SUBAPPLICATION logiBUS_AI_Calibrate_3P_Subscribe_VT_OPC (* Remote-Subscribe eines bereits kalibrierten physikalischen Werts (M2M, von der Sensor-Station, 3-Punkt-Kalibrierung) -> VT-Anzeige (Q_NumericValue_PHYSA) + lokaler Re-Publish + optionaler CAL_OUT-Plug fuer lokale Consumer. Die physischen VT-Elemente bleiben hier (dort wo die VT ist): C_MIN/C_MID/C_MAX-Tasten rufen per CLIENT_0 direkt die ID_MIN_METHOD/ID_MID_TRIGGER_METHOD/ID_MAX_METHOD auf der Sensor-Station auf (logiBUS_AI_Calibrate_3P_IDA_OPC) - echter Event-zu-Event-Methodenaufruf, kein Toggle/Publish/Subscribe-Umweg. Die drei Referenzwert-Eingabefelder MIN/MID/MAX_REF (NumericValue_TO_AR2_OPC) werden weiterhin LOKAL publiziert und von der Sensor-Station remote abonniert - MID_REF/MAX_REF zusaetzlich als plain-AR-Plugs MIDREF_OUT/MAXREF_OUT re-exponiert (z.B. fuer Fuellband_Oben_Erkennung/Befuellautomatik). Ersetzt logiBUS_AI_Calibrate_3P_Remote_IDA_OPC: Kalibrierung selbst laeuft jetzt auf der Sensor-Station (logiBUS_AI_Calibrate_3P_IDA_OPC), hier bleibt nur noch Anzeige + VT-Bedienelemente-Weiterleitung. *)
  (* Standard: 61499-2; Description: Copyright (c) 2026 Meisterschulen am Ostbahnhof This program and the accompanying materials are made available under the terms of the Eclipse Public License 2.0 which is available at https://www.eclipse.org/legal/epl-2.0/ SPDX-License-Identifier: EPL-2.0 *)
  (* Version 1.0, 2026-09-18, Franz Höpfinger, Meisterschulen am Ostbahnhof, initial implementation - Analog-Lokal-Verarbeitung Phase 6 (Plan cuddly-bubbling-twilight): 3P-Pendant zu logiBUS_AI_Calibrated_Subscribe_VT_OPC (2P), fuer Fuellband Winkel (STG2). Plugs CAL_OUT/MIDREF_OUT/MAXREF_OUT 1:1 aus logiBUS_AI_Calibrate_3P_Remote_IDA_OPC uebernommen, damit bestehende Consumer (Fuellband_Oben_Erkennung, Befuellautomatik) unveraendert bleiben. *)
  PACKAGE MyLib::sys;
  IMPORT isobus::UT::Q::const::IDs::ID_NULL;
  IMPORT isobus::UT::io::Button::ButtonActivationCode::BT_PRESSED_LATCHED;
  IMPORT logiBUS::utils::conversion::phys::NumericObjectPool_S;
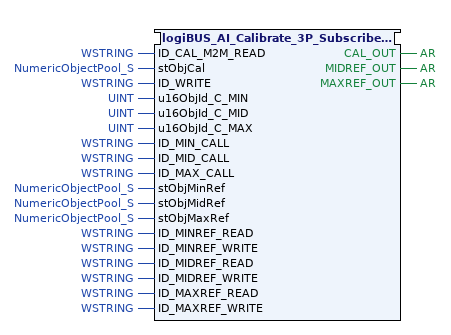
  VAR_INPUT
    ID_CAL_M2M_READ : WSTRING; (* Remote-Subscribe-Adresse des bereits kalibrierten physikalischen Werts (REAL) - Gegenstueck zu ID_CAL_WRITE auf der Sensor-Station (logiBUS_AI_Calibrate_3P_IDA_OPC) *)
    stObjCal : logiBUS::utils::conversion::phys::NumericObjectPool_S := (u16ObjId := ID_NULL, r32Scale := 1.0, i32Offset := 0, u8Decimals := 1); (* Object ID + Scale/Offset/Decimals CNumberVariable (kalibrierter Wert) *)
    ID_WRITE : WSTRING; (* Lokale Re-Publish-Adresse (REAL, ACTION=PUBLISH) fuer weitere lokale Konsumenten auf dieser Station *)
    u16ObjId_C_MIN : UINT := ID_NULL; (* Object ID Taste 'C_MIN' - physisch hier auf der VT *)
    u16ObjId_C_MID : UINT := ID_NULL; (* Object ID Taste 'C_MID' - physisch hier auf der VT *)
    u16ObjId_C_MAX : UINT := ID_NULL; (* Object ID Taste 'C_MAX' - physisch hier auf der VT *)
    ID_MIN_CALL : WSTRING; (* Remote-Methodenadresse (ACTION=CALL_METHOD) fuer den C_MIN-Trigger - ruft ID_MIN_METHOD direkt auf der Sensor-Station auf (logiBUS_AI_Calibrate_3P_IDA_OPC) *)
    ID_MID_CALL : WSTRING; (* Remote-Methodenadresse (ACTION=CALL_METHOD) fuer den C_MID-Trigger - ruft ID_MID_TRIGGER_METHOD direkt auf der Sensor-Station auf *)
    ID_MAX_CALL : WSTRING; (* Remote-Methodenadresse (ACTION=CALL_METHOD) fuer den C_MAX-Trigger - ruft ID_MAX_METHOD direkt auf der Sensor-Station auf *)
    stObjMinRef : logiBUS::utils::conversion::phys::NumericObjectPool_S := (u16ObjId := ID_NULL, r32Scale := 1.0, i32Offset := 0, u8Decimals := 1); (* Object ID + Scale/Offset/Decimals CNumberVariable (MIN_REF-Referenzwert, VT-Eingabefeld hier auf dieser Station) *)
    stObjMidRef : logiBUS::utils::conversion::phys::NumericObjectPool_S := (u16ObjId := ID_NULL, r32Scale := 1.0, i32Offset := 0, u8Decimals := 1); (* Object ID + Scale/Offset/Decimals CNumberVariable (MID_REF-Referenzwert, VT-Eingabefeld hier auf dieser Station) *)
    stObjMaxRef : logiBUS::utils::conversion::phys::NumericObjectPool_S := (u16ObjId := ID_NULL, r32Scale := 1.0, i32Offset := 0, u8Decimals := 1); (* Object ID + Scale/Offset/Decimals CNumberVariable (MAX_REF-Referenzwert, VT-Eingabefeld hier auf dieser Station) *)
    ID_MINREF_READ : WSTRING; (* Optionale Subscribe-Adresse falls MIN_REF extern (Dashboard) ueberschrieben werden soll - unbenutzt zulaessig *)
    ID_MINREF_WRITE : WSTRING; (* Lokale Publish-Adresse (REAL, ACTION=PUBLISH) des MIN_REF-Referenzwerts - wird von der Sensor-Station remote abonniert (deren ID_MINREF_READ) *)
    ID_MIDREF_READ : WSTRING; (* Optionale Subscribe-Adresse falls MID_REF extern (Dashboard) ueberschrieben werden soll - unbenutzt zulaessig *)
    ID_MIDREF_WRITE : WSTRING; (* Lokale Publish-Adresse (REAL, ACTION=PUBLISH) des MID_REF-Referenzwerts - wird von der Sensor-Station remote abonniert (deren ID_MIDREF_READ) *)
    ID_MAXREF_READ : WSTRING; (* Optionale Subscribe-Adresse falls MAX_REF extern (Dashboard) ueberschrieben werden soll - unbenutzt zulaessig *)
    ID_MAXREF_WRITE : WSTRING; (* Lokale Publish-Adresse (REAL, ACTION=PUBLISH) des MAX_REF-Referenzwerts - wird von der Sensor-Station remote abonniert (deren ID_MAXREF_READ) *)
  END_VAR
  PLUGS
    CAL_OUT : adapter::types::unidirectional::AR; (* Optional: kalibrierter Wert (plain-AR-Spiegel des Remote-Subscribe) fuer externe lokale Consumer, statt eigenem lokalen OPC-UA-Self-Subscribe. Unverdrahtet lassen, wenn nicht gebraucht. *)
    MIDREF_OUT : adapter::types::unidirectional::AR; (* Optional: live MID_REF-Referenzwert (= MID_REF_LIT.VALUE_OUT) fuer externe Consumer. Unverdrahtet lassen, wenn nicht gebraucht. *)
    MAXREF_OUT : adapter::types::unidirectional::AR; (* Optional: live MAX_REF-Referenzwert (= MAX_REF_LIT.VALUE_OUT) fuer externe Consumer. Unverdrahtet lassen, wenn nicht gebraucht. *)
  END_PLUGS
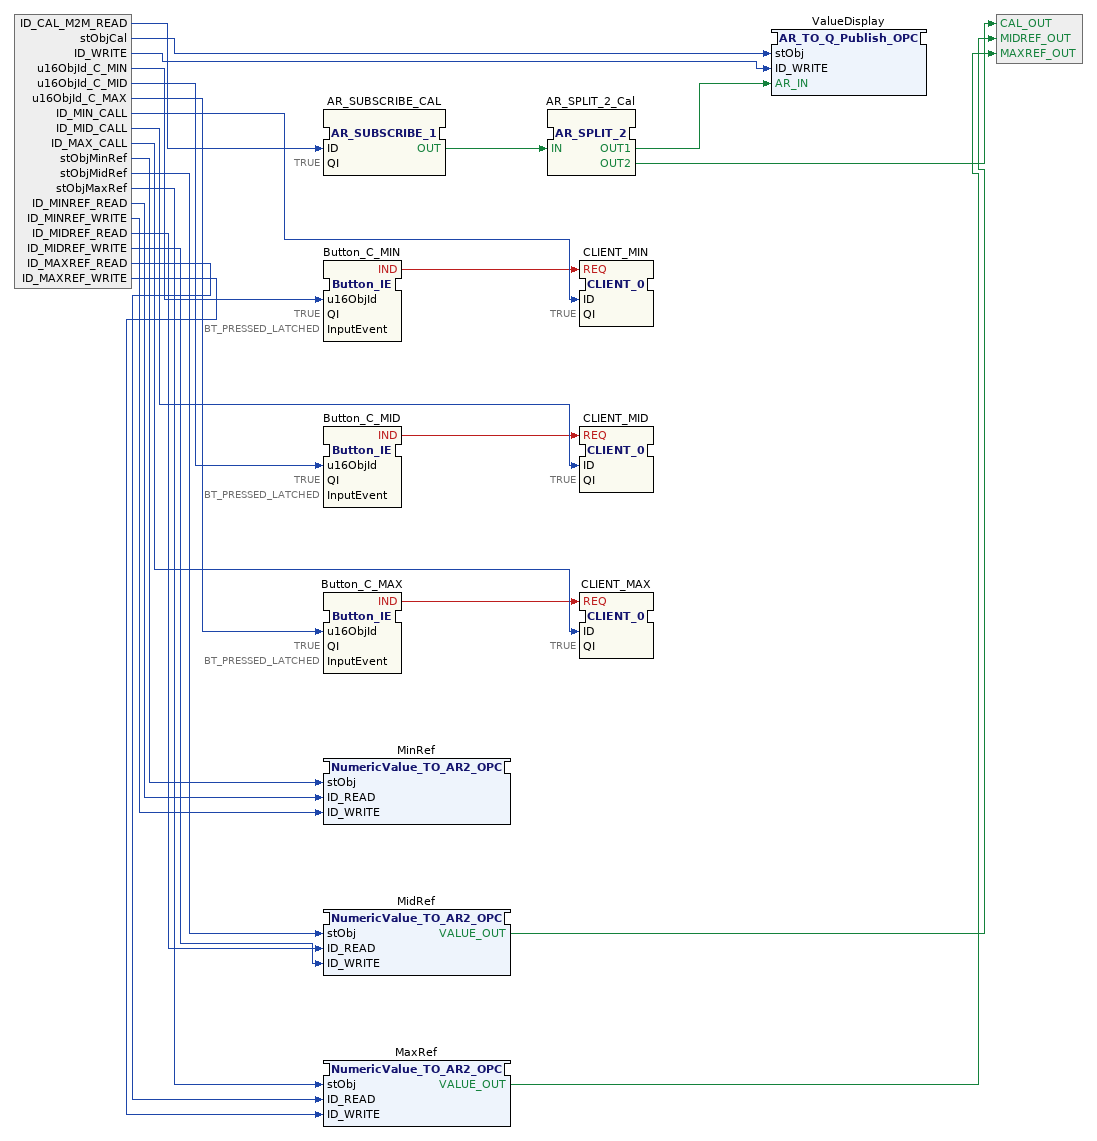
  FBS
    AR_SUBSCRIBE_CAL : adapter::net::AR_SUBSCRIBE_1(QI := TRUE);
    AR_SPLIT_2_Cal : adapter::events::unidirectional::AR_SPLIT_2;
    Button_C_MIN : isobus::UT::io::Button::Button_IE(QI := TRUE, InputEvent := BT_PRESSED_LATCHED);
    Button_C_MID : isobus::UT::io::Button::Button_IE(QI := TRUE, InputEvent := BT_PRESSED_LATCHED);
    Button_C_MAX : isobus::UT::io::Button::Button_IE(QI := TRUE, InputEvent := BT_PRESSED_LATCHED);
    CLIENT_MIN : iec61499::net::CLIENT_0(QI := TRUE);
    CLIENT_MID : iec61499::net::CLIENT_0(QI := TRUE);
    CLIENT_MAX : iec61499::net::CLIENT_0(QI := TRUE);
  END_FBS
  SUBAPPS
    ValueDisplay : MyLib::sys::AR_TO_Q_Publish_OPC;
    MinRef : MyLib::sys::NumericValue_TO_AR2_OPC;
    MidRef : MyLib::sys::NumericValue_TO_AR2_OPC;
    MaxRef : MyLib::sys::NumericValue_TO_AR2_OPC;
  END_SUBAPPS
  EVENT_CONNECTIONS
    Button_C_MIN.IND TO CLIENT_MIN.REQ;
    Button_C_MID.IND TO CLIENT_MID.REQ;
    Button_C_MAX.IND TO CLIENT_MAX.REQ;
  END_CONNECTIONS
  DATA_CONNECTIONS
    ID_CAL_M2M_READ TO AR_SUBSCRIBE_CAL.ID;
    stObjCal TO ValueDisplay.stObj;
    ID_WRITE TO ValueDisplay.ID_WRITE;
    u16ObjId_C_MIN TO Button_C_MIN.u16ObjId;
    u16ObjId_C_MID TO Button_C_MID.u16ObjId;
    u16ObjId_C_MAX TO Button_C_MAX.u16ObjId;
    ID_MIN_CALL TO CLIENT_MIN.ID;
    ID_MID_CALL TO CLIENT_MID.ID;
    ID_MAX_CALL TO CLIENT_MAX.ID;
    stObjMinRef TO MinRef.stObj;
    ID_MINREF_READ TO MinRef.ID_READ;
    ID_MINREF_WRITE TO MinRef.ID_WRITE;
    stObjMidRef TO MidRef.stObj;
    ID_MIDREF_READ TO MidRef.ID_READ;
    ID_MIDREF_WRITE TO MidRef.ID_WRITE;
    stObjMaxRef TO MaxRef.stObj;
    ID_MAXREF_READ TO MaxRef.ID_READ;
    ID_MAXREF_WRITE TO MaxRef.ID_WRITE;
  END_CONNECTIONS
  ADAPTER_CONNECTIONS
    AR_SUBSCRIBE_CAL.OUT TO AR_SPLIT_2_Cal.IN;
    AR_SPLIT_2_Cal.OUT1 TO ValueDisplay.AR_IN;
    AR_SPLIT_2_Cal.OUT2 TO CAL_OUT;
    MidRef.VALUE_OUT TO MIDREF_OUT;
    MaxRef.VALUE_OUT TO MAXREF_OUT;
  END_CONNECTIONS
END_SUBAPPLICATION
